TYPE ST_CameraPara :
STRUCT
	tDelay:TIME;
END_STRUCT
END_TYPE

(* stored: Version 1.1.0.1, ProductVersion 3.1.4024.9
   DUT ST_CameraPara: Id {5fe6a014-db5c-463b-a4c7-e3e598e81ee3} *)
